FUNCTION_BLOCK BYTE2BYTE
  {SET_ATTRIBUTE(OpcUa, SERVICE)}
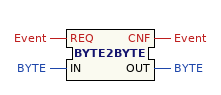
  EVENT_INPUT
    REQ;
  END_EVENT
  EVENT_OUTPUT
    CNF;
  END_EVENT
  VAR_INPUT
    IN : BYTE;
  END_VAR
  VAR_OUTPUT
    OUT : BYTE;
  END_VAR
END_FUNCTION_BLOCK
